# B&R Automation Studio project ZariadenieNaPreklapanieRotorov
Automation Studio 4.7.6.114 SP; Default project

## Configuration Config1

CPU 4PPC30.043F-21B, AutomationRuntime D4.73, Build 6.3.0, Vc V4.72.5

### Task classes (Cpu.sw)
```
Cyclic#3 (cycle 50000 us, tolerance 50000 us):
  Blikanie10 <- Blikace.Blikanie100ms.prg
Cyclic#4 (cycle 100000 us, tolerance 100000 us):
  Blikanie20 <- Blikace.Blikanie200ms.prg
  DatumCasPL <- DatumCasPLC.DatumCasPLC.prg
  Main <- Program.Main.prg
  Preklapac <- Program.Preklapac.prg
  Alarmy <- Program.Alarmy.prg
  OvladanieV <- HMI.OvladanieVizu.prg
Cyclic#5 (cycle 250000 us, tolerance 250000 us):
  Blikanie50 <- Blikace.Blikanie500ms.prg
Cyclic#7 (cycle 1000000 us, tolerance 1000000 us):
  Blikanie1s <- Blikace.Blikanie1s.prg
VcDataObjects: Visu <- HMI.Visu.dob
Binaries: vcctext, arialbd, vccshape, vcchspot, vcnet, vcdsloc, vcbclass, vcfntttf, vccovl, vctcal, Visu03, vcshared, vcpd335x, vcpkat, vcpk, vccbmp, TCData, vcfile, vccbtn, vcmgr, vccdt, vcptelo, vcalarm, Visu01, vccnum, vcpdsw, FWRules, vcrt, arial, udbdef, vcpfppct, vcgclass, vcpdvnc, vccalarm, vccstr, vcdsint, vccbar, Visu02, Role, arconfig, User, asfw, ashwd, ashwac, sysconf, iomap
Libraries: IecCheck, SC, sys_lib, AsBrStr, Runtime, asieccon, fileio, dataobj, astime, standard, vcresman
```

### Hardware
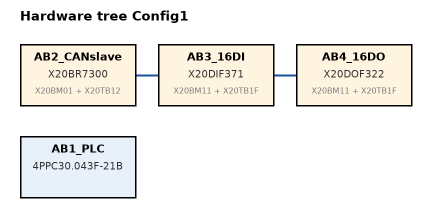
```
AB1_PLC : 4PPC30.043F-21B v1.1.3.0
  Connector IF3:
    ActivateDevice = 1
    Mode = Manual
    InternetAddress = 192.168.1.2
    SubnetMask = 255.255.255.0
    InaNodeNumber = 0
    Vnc1
    VncVcObjectName1 = Visu
    VncKeyMappingFile1 = VC\PS2-Keyboard.dis
    VncMaxConnections1 = 2
    VncRefreshRate1 = 100
  ConfigurationID = ZariadenieNaPreklapanieRotorov_Config1
  PermanentPvSize = 500
  TimerDeviceType = SWIOTIMER
  Cyclic1Duration = 1000
  Cyclic1Tolerance = 0
  Cyclic2Duration = 20000
  Cyclic2Tolerance = 20000
  Cyclic3Duration = 50000
  Cyclic3Tolerance = 50000
  Cyclic4Duration = 100000
  Cyclic4Tolerance = 100000
  Cyclic5Duration = 250000
  Cyclic5Tolerance = 250000
  Cyclic6Duration = 500000
  Cyclic6Tolerance = 500000
  Cyclic7Duration = 1000000
  Cyclic7Tolerance = 1000000
  Cyclic8Duration = 10000
  Cyclic8Tolerance = 30000000
  TimeZone = 145
  VcObjectName = Visu
  RotationAngle = 180
  KeyMappingFile = VC\4PPC30_043F_21B.dis
AB2_CANslave : X20BR7300 v1.4.0.0  [CAN1 -> AB1_PLC.IF4; SL -> X20BM01.SL1; SS1 -> X20TB12.SS]
  Supervision = off
AB3_16DI : X20DIF371 v1.1.0.0  [SS1 -> X20TB1F.SS; SL -> X20BM11.SL1]
  FunctionModel = CANIOBusController
  Supervision = off
AB4_16DO : X20DOF322 v1.4.0.0  [SS1 -> X20TB1F1.SS; SL -> X20BM11a.SL1]
  FunctionModel = CANIOBusController
  Supervision = off
X20BM01 : X20BM01 v2.1.0.0
X20BM11 : X20BM11 v1.0.0.1  [X2X1 -> X20BM01.IF1]
X20BM11a : X20BM11 v1.0.0.1  [X2X1 -> X20BM11.X2X2]
X20TB12 : X20TB12 v1.0.0.0
X20TB1F : X20TB1F v1.0.0.0
X20TB1F1 : X20TB1F v1.0.0.0
```

### IoMap.iom - AB1_PLC/IoMap.iom
```iecst
VAR_CONFIG
	Hardware.KartaAB2_CANSlave_OK AT %IX."AB2_CANslave".IF1.ST1.ModuleOk;
	Hardware.KartaAB3_16DI_OK AT %IX."AB3_16DI".ModuleOk;
	Hardware.KartaAB4_16DO_OK AT %IX."AB4_16DO".ModuleOk;
	Cyclic#1.Zariadenie.IN.TlakVzduchu_OK_S1 AT %IX."AB3_16DI".DigitalInput01;
	Cyclic#1.Preklapac.IN.VstupnyDotlacac_VYSUNUTY_MS1 AT %IX."AB3_16DI".DigitalInput02;
	Cyclic#1.Preklapac.IN.VstupnyDotlacac_ZASUNUTY_MS2 AT %IX."AB3_16DI".DigitalInput03;
	Cyclic#1.Preklapac.IN.VystupnyDotlacac_VYSUNUTY_MS3 AT %IX."AB3_16DI".DigitalInput04;
	Cyclic#1.Preklapac.IN.VystupnyDotlacac_ZASUNUTY_MS4 AT %IX."AB3_16DI".DigitalInput05;
	Cyclic#1.Preklapac.IN.Vytah_HornaPoloha_MS5 AT %IX."AB3_16DI".DigitalInput06;
	Cyclic#1.Preklapac.IN.Vytah_SpodnaPoloha_MS6 AT %IX."AB3_16DI".DigitalInput07;
	Cyclic#1.Preklapac.IN.VstupnyDotlacac_PritomRotora_IS1 AT %IX."AB3_16DI".DigitalInput08;
	Cyclic#1.Zariadenie.IN.Safety_SpatnaVazba_KF1 AT %IX."AB3_16DI".DigitalInput09;
	Cyclic#1.Preklapac.IN.Vytah_Pozicia1_PritomRotora_OS1 AT %IX."AB3_16DI".DigitalInput11;
	Cyclic#1.Preklapac.IN.Vytah_Pozicia2_PritomRotora_OS2 AT %IX."AB3_16DI".DigitalInput12;
	Cyclic#1.Preklapac.IN.VystupnyDopravnik_PLNY_OS3 AT %IX."AB3_16DI".DigitalInput13;
	Cyclic#1.Zariadenie.OUT.Majak_ZeleneSvetlo AT %QX."AB4_16DO".DigitalOutput01;
	Cyclic#1.Zariadenie.OUT.Majak_ZlteSvetlo AT %QX."AB4_16DO".DigitalOutput02;
	Cyclic#1.Zariadenie.OUT.Majak_CerveneSvetlo AT %QX."AB4_16DO".DigitalOutput03;
	Cyclic#1.Zariadenie.OUT.Majak_Hukacka AT %QX."AB4_16DO".DigitalOutput04;
	Cyclic#1.Zariadenie.OUT.Safety_RESET AT %QX."AB4_16DO".DigitalOutput05;
	Cyclic#1.Preklapac.OUT.VstupnyDotlacac_VYSUN_YV1 AT %QX."AB4_16DO".DigitalOutput06;
	Cyclic#1.Preklapac.OUT.VstupnyDotlacac_ZASUN_YV2 AT %QX."AB4_16DO".DigitalOutput07;
	Cyclic#1.Preklapac.OUT.VystupnyDotlacac_VYSUN_YV3 AT %QX."AB4_16DO".DigitalOutput08;
	Cyclic#1.Preklapac.OUT.Vytah_ZDVIH_YV5 AT %QX."AB4_16DO".DigitalOutput10;
	Cyclic#1.Preklapac.OUT.Vytah_ZOSTUP_YV6 AT %QX."AB4_16DO".DigitalOutput11;
	Cyclic#1.Zariadenie.IN.Safety_SpatnaVazba_Ventil_YVS1 AT %IX."AB3_16DI".DigitalInput14;
	Cyclic#1.Zariadenie.IN.Safety_SpatnaVazba_Ventil_YVS2 AT %IX."AB3_16DI".DigitalInput15;
	Cyclic#1.Zariadenie.IN.Safety_Aktivne AT %IX."AB3_16DI".DigitalInput16;
	Cyclic#1.Preklapac.IN.VystupnyDopravnik_StavOK AT %IX."AB3_16DI".DigitalInput10;
END_VAR
```

- Physical/Config1/AB1_PLC/PvMap.vvm: same as Physical/Config1/AB1_PLC/Cpu.per
## Logical view

Binary libraries used (declarations not repeated): RUNTIME, OPERATOR, AsIecCon, astime, standard, AsBrStr, FileIO, sys_lib

### Global.typ - Global data types
```iecst
(********************************************************************
 * COPYRIGHT -- Microsoft
 ********************************************************************
 * File: Global.typ
 * Author: Martin
 * Created: February 11, 2016
 ********************************************************************
 * Global data types of project Zamazat_1
 ********************************************************************)
(**************Stav hardware*****************************)

TYPE
	HardwareSTAV_typ : 	STRUCT
		KartaAB2_CANSlave_OK : BOOL;
		KartaAB3_16DI_OK : BOOL;
		KartaAB4_16DO_OK : BOOL;
	END_STRUCT;
END_TYPE

(**************************Vizualizacia**********************************************)

TYPE
	Vizu_typ : 	STRUCT
		CisloAktualnejObrazovky : USINT;
		CisloZadanejObrazovky : USINT;
		TL_RezimAutomat : BOOL;
		StavZariadenia_Farba : USINT;
		StavZariadenia_Index : USINT;
		TL_RezimManual_DISABLE : BOOL; (*0 - odomknuté, 1 - zamknuté*)
		TL_StartAutomat_DISABLE : BOOL;
		TL_UkoncenieCyklu_DISABLE : BOOL;
		TL_Reset_DISABLE : BOOL;
		TL_RR_PreklapacDotlacace_DISABLE : BOOL;
		TL_RR_PreklapacZdvih_DISABLE : BOOL;
		Slider : USINT;
		FarbaTlacitkaAlarm_Index : BOOL;
		ZobrazSymbolAlarmu : BOOL;
		TP_PopUp_ResetZariadenia : USINT;
		TP_PopUp_VystupDopRozpojeny : USINT;
		PodsvietenieTlacitka_ResetCS : USINT;
	END_STRUCT;
END_TYPE

(**************************Pracovisko************************************************)

TYPE
	Zariadenie_typ : 	STRUCT
		IN : ZariadenieIN_typ;
		OUT : ZariadenieOUT_typ;
		PAR : ZariadeniePAR_typ;
		STAV : ZariadenieSTAV_typ;
		Automat : BOOL;
		Manual : BOOL;
		Reset : BOOL;
		KoniecCyklu : BOOL;
		Majak_HukackaON : BOOL;
	END_STRUCT;
	ZariadenieIN_typ : 	STRUCT
		TlakVzduchu_OK_S1 : BOOL;
		Safety_SpatnaVazba_KF1 : BOOL;
		Safety_ReleCakaNaReset_KF1 : BOOL;
		Safety_SpatnaVazba_Ventil_YVS1 : BOOL;
		Safety_SpatnaVazba_Ventil_YVS2 : BOOL;
		Safety_Aktivne : BOOL;
	END_STRUCT;
	ZariadenieOUT_typ : 	STRUCT
		Majak_ZeleneSvetlo : BOOL;
		Majak_ZlteSvetlo : BOOL;
		Majak_CerveneSvetlo : BOOL;
		Majak_Hukacka : BOOL;
		Safety_RESET : BOOL;
	END_STRUCT;
	ZariadeniePAR_typ : 	STRUCT
		PAR_0 : USINT;
	END_STRUCT;
	ZariadenieSTAV_typ : 	STRUCT
		Automat : BOOL;
		Manual : BOOL;
		PoINIT : BOOL;
		READY_TO_START : BOOL;
		UkoncenieCyklu_BUSY : BOOL;
		Hardware_OK : BOOL;
	END_STRUCT;
END_TYPE

(***************Preklapač*************************************)

TYPE
	Preklapac_typ : 	STRUCT
		IN : PreklapacIN_typ;
		OUT : PreklapacOUT_typ;
		PAR : PreklapacPAR_typ;
		STAV : PreklapacSTAV_typ;
		Automat : BOOL;
		Manual : BOOL;
		Reset : BOOL;
		KoniecCyklu : BOOL;
	END_STRUCT;
	PreklapacIN_typ : 	STRUCT
		VstupnyDotlacac_VYSUNUTY_MS1 : BOOL;
		VstupnyDotlacac_ZASUNUTY_MS2 : BOOL;
		VstupnyDotlacac_PritomRotora_IS1 : BOOL;
		VystupnyDotlacac_VYSUNUTY_MS3 : BOOL;
		VystupnyDotlacac_ZASUNUTY_MS4 : BOOL;
		Vytah_HornaPoloha_MS5 : BOOL;
		Vytah_SpodnaPoloha_MS6 : BOOL;
		Vytah_Pozicia1_PritomRotora_OS1 : BOOL;
		Vytah_Pozicia2_PritomRotora_OS2 : BOOL;
		VystupnyDopravnik_PLNY_OS3 : BOOL;
		VystupnyDopravnik_StavOK : BOOL;
	END_STRUCT;
	PreklapacOUT_typ : 	STRUCT
		VstupnyDotlacac_VYSUN_YV1 : BOOL;
		VstupnyDotlacac_ZASUN_YV2 : BOOL;
		VystupnyDotlacac_VYSUN_YV3 : BOOL;
		Vytah_ZDVIH_YV5 : BOOL;
		Vytah_ZOSTUP_YV6 : BOOL;
	END_STRUCT;
	PreklapacPAR_typ : 	STRUCT
		PAR_0 : USINT;
	END_STRUCT;
	PreklapacSTAV_typ : 	STRUCT
		PoINIT : BOOL;
	END_STRUCT;
END_TYPE
```

### Global.var - Global variables
```iecst
(********************************************************************
 * COPYRIGHT -- Microsoft
 ********************************************************************
 * File: Global.var
 * Author: Martin
 * Created: February 11, 2016
 ********************************************************************
 * Global variables of project Zamazat_1
 ********************************************************************)
(******************Blikače*****************************)
VAR
	Blikac100ms : BOOL;
	Blikac200ms : BOOL;
	Blikac500ms : BOOL;
	Blikac1s : BOOL;
END_VAR
(**********Nastavenie času**************)
VAR
	DTSetTime_0 : DTSetTime := (0);
	DTGetTime_0 : DTGetTime := (0);
END_VAR
(*****************Alarmy*****************************)
VAR
	Alarmy : ARRAY[0..100] OF BOOL;
	NastalaPorucha : BOOL;
	PotvrdenieAlarmov : BOOL;
END_VAR
(*************Všeobecné premenné*************)
VAR
	Hardware : HardwareSTAV_typ := (0);
	Zariadenie : Zariadenie_typ := (0);
	Vizu : Vizu_typ := (0);
	Preklapac : Preklapac_typ := (0);
	SC_Preklapac : SequenceControlTyp := (0);
END_VAR
```

### Package Logical/Libraries - Global libraries

### Library Logical/Libraries/SC (IEC)

#### Types.typ - Exported data types
```iecst
TYPE
	SequenceControlTyp : 	STRUCT
		StepName : STRING[200];
		Step : UINT;
		Switch1 : BOOL;
		Switch2 : BOOL;
		Switch3 : BOOL;
		ResetStep : BOOL;
		LastStep : BOOL;
		IdleTime : TON;
		AlarmTime : TON;
	END_STRUCT;
END_TYPE
```

#### SC.fun - Exported functions and function blocks
```iecst
FUNCTION SequenceControl : BOOL
	VAR_IN_OUT
		SC : SequenceControlTyp;
	END_VAR
END_FUNCTION
```

#### SequenceControl.st
```iecst
(* TODO: Add your comment here *)
FUNCTION SequenceControl

	IF SC.ResetStep THEN
		brsmemset(ADR(SC.StepName),0,SIZEOF(SC.StepName));
		SC.Switch1:= FALSE;
		SC.Switch2:= FALSE;
		SC.Switch3:= FALSE;
		SC.IdleTime.IN:= FALSE;
		SC.AlarmTime.IN:= FALSE;
		SC.ResetStep:= FALSE;
	END_IF

	IF SC.LastStep THEN
		brsmemset(ADR(SC.StepName),0,SIZEOF(SC.StepName));
		SC.Switch1:= FALSE;
		SC.Switch2:= FALSE;
		SC.Switch3:= FALSE;
		SC.IdleTime.IN:= FALSE;
		SC.AlarmTime.IN:= FALSE;
		SC.Step:= 0;
		SC.LastStep:= FALSE;
	END_IF

	//Volanie časovačov//
	SC.AlarmTime();
	SC.IdleTime();

END_FUNCTION
```

### Library Logical/Libraries/IecCheck (IEC)
Depends on: sys_lib, AsBrStr

#### IecCheck.fun - Exported functions and function blocks
```iecst
FUNCTION CheckDivSint : SINT (* Check divisor for SINT division *)
	VAR_INPUT
		divisor : SINT;
	END_VAR
END_FUNCTION

FUNCTION CheckDivUsint : USINT (* Check divisor for USINT division *)
	VAR_INPUT
		divisor : USINT;
	END_VAR
END_FUNCTION

FUNCTION CheckDivInt : INT (* Check divisor for INT division *)
	VAR_INPUT
		divisor : INT;
	END_VAR
END_FUNCTION

FUNCTION CheckDivUint : UINT (* Check divisor for UINT division *)
	VAR_INPUT
		divisor : UINT;
	END_VAR
END_FUNCTION

FUNCTION CheckDivDint : DINT (* Check divisor for DINT division *)
	VAR_INPUT
		divisor : DINT;
	END_VAR
END_FUNCTION

FUNCTION CheckDivUdint : UDINT (* Check divisor for UDINT division *)
	VAR_INPUT
		divisor : UDINT;
	END_VAR
END_FUNCTION

FUNCTION CheckDivReal : REAL (* Check divisor for REAL division *)
	VAR_INPUT
		divisor : REAL;
	END_VAR
END_FUNCTION

FUNCTION CheckDivLReal : LREAL (* Check divisor for LREAL division, not available for SG3 and SGC *)
	VAR_INPUT
		divisor : LREAL;
	END_VAR
END_FUNCTION

FUNCTION CheckBounds : DINT (* Check range for array access *)
	VAR_INPUT
		index : DINT;
		lower : DINT;
		upper : DINT;
	END_VAR
END_FUNCTION

FUNCTION CheckRange : DINT (* Check range for enumeration *)
	VAR_INPUT
		value : DINT;
		lower : DINT;
		upper : DINT;
	END_VAR
END_FUNCTION

FUNCTION CheckSignedSubrange : DINT (* Check range for subrange of signed data types *)
	VAR_INPUT
		value : DINT;
		lower : DINT;
		upper : DINT;
	END_VAR
END_FUNCTION

FUNCTION CheckUnsignedSubrange : UDINT (* Check range for subrange of unsigned data types *)
	VAR_INPUT
		value : UDINT;
		lower : UDINT;
		upper : UDINT;
	END_VAR
END_FUNCTION

FUNCTION CheckReadAccess : UDINT (* Check address when reading dynamic variables *)
	VAR_INPUT
		address : UDINT;
	END_VAR
END_FUNCTION

FUNCTION CheckWriteAccess : UDINT (* Check address when writing dynamic variables *)
	VAR_INPUT
		address : UDINT;
	END_VAR
END_FUNCTION

FUNCTION MakeEntry : UDINT (* Makes an entry (log book entry) in the error log book *)
	VAR
		taskname : STRING[30];
		group : USINT;
		status_name : UINT;
		out_text : STRING[80];
	END_VAR
	VAR_INPUT
		number : UINT;
		index : DINT;
		text : STRING[50];
	END_VAR
END_FUNCTION
```

#### IecCheck.st - Implementation file
```iecst
(* Check divisor for SINT division *)
FUNCTION CheckDivSint
	IF divisor=0 THEN
		CheckDivSint:=1;
		MakeEntry(55555,divisor,'CheckDivSint');
	ELSE
		CheckDivSint:=divisor;
	END_IF
END_FUNCTION

(* Check divisor for USINT division *)
FUNCTION CheckDivUsint
	IF divisor=0 THEN
		CheckDivUsint:=1;
		MakeEntry(55555,divisor,'CheckDivUsint');
	ELSE
		CheckDivUsint:=divisor;
	END_IF
END_FUNCTION

(* Check divisor for INT division *)
FUNCTION CheckDivInt
	IF divisor=0 THEN
		CheckDivInt:=1;
		MakeEntry(55555,divisor,'CheckDivInt');
	ELSE
		CheckDivInt:=divisor;
	END_IF
END_FUNCTION

(* Check divisor for UINT division *)
FUNCTION CheckDivUint
	IF divisor=0 THEN
		CheckDivUint:=1;
		MakeEntry(55555,divisor,'CheckDivUint');
	ELSE
		CheckDivUint:=divisor;
	END_IF
END_FUNCTION

(* Check divisor for DINT division *)
FUNCTION CheckDivDint
	IF divisor=0 THEN
		CheckDivDint:=1;
		MakeEntry(55555,divisor,'CheckDivDint');
	ELSE
		CheckDivDint:=divisor;
	END_IF
END_FUNCTION

(* Check divisor for UDINT division *)
FUNCTION CheckDivUdint
	IF divisor=0 THEN
		CheckDivUdint:=1;
		MakeEntry(55555,divisor,'CheckDivUdint');
	ELSE
		CheckDivUdint:=divisor;
	END_IF
END_FUNCTION

(* Check divisor for REAL division *)
FUNCTION CheckDivReal
	IF divisor=0 THEN
		CheckDivReal:=1;
		MakeEntry(55555,0,'CheckDivReal');
	ELSE
		CheckDivReal:=divisor;
	END_IF
END_FUNCTION

(* Check divisor for LREAL division *)
FUNCTION CheckDivLReal
	IF divisor=0 THEN
		CheckDivLReal:=1;
		MakeEntry(55555,0,'CheckDivLReal');
	ELSE
		CheckDivLReal:=divisor;
	END_IF
END_FUNCTION

(* Check range for array access *)
FUNCTION CheckBounds
	IF index < lower THEN
		CheckBounds := lower;
		MakeEntry(55555,index,'CheckBounds');
	ELSIF index > upper THEN
		CheckBounds := upper;
		MakeEntry(55555,index,'CheckBounds');
	ELSE
		CheckBounds := index;
	END_IF
END_FUNCTION

(* Check range for enumeration *)
FUNCTION CheckRange
	IF value < lower THEN
		CheckRange := lower;
		MakeEntry(55555,value,'CheckRange');
	ELSIF value > upper THEN
		CheckRange := upper;
		MakeEntry(55555,value,'CheckRange');
	ELSE
		CheckRange := value;
	END_IF
END_FUNCTION

(* Check range for subrange of signed data types *)
FUNCTION CheckSignedSubrange
	IF value < lower THEN
		CheckSignedSubrange := lower;
		MakeEntry(55555,value,'CheckSignedSubrange');
	ELSIF value > upper THEN
		CheckSignedSubrange := upper;
		MakeEntry(55555,value,'CheckSignedSubrange');
	ELSE
		CheckSignedSubrange := value;
	END_IF
END_FUNCTION

(* Check range for subrange of unsigned data types *)
FUNCTION CheckUnsignedSubrange
	IF value < lower THEN
		CheckUnsignedSubrange := lower;
		MakeEntry(55555,value,'CheckUnsignedSubrange');
	ELSIF value > upper THEN
		CheckUnsignedSubrange := upper;
		MakeEntry(55555,value,'CheckUnsignedSubrange');
	ELSE
		CheckUnsignedSubrange := value;
	END_IF
END_FUNCTION

(* Check address when reading dynamic variables *)
FUNCTION CheckReadAccess
	IF address=0 THEN
		(* TODO: Insert an appropriate code, see AutomationStudio help for further information *)
		MakeEntry(55555,address,'Read from NULL');
	END_IF

	CheckReadAccess:=0;
END_FUNCTION

(* Check address when writing dynamic variables *)
FUNCTION CheckWriteAccess
	IF address=0 THEN
		(* TODO: Insert an appropriate code, see AutomationStudio help for further information *)
		MakeEntry(55555,address,'Write to NULL');
	END_IF

	CheckWriteAccess:=0;
END_FUNCTION

(* Makes an entry (log book entry) in the error log book *)
FUNCTION MakeEntry
		status_name := ST_name(0,ADR(taskname),ADR(group));

		brsstrcpy(ADR(out_text),ADR(text));
		brsstrcat(ADR(out_text),ADR(' > in task > '));
  		brsstrcat(ADR(out_text),ADR(taskname));
		MakeEntry := ADR(out_text);
		ERRxfatal(number,index,ADR(out_text));
END_FUNCTION
```

### Package Logical/Program - Riadiace programy

### Program Logical/Program/Main (IEC)

#### Main.st - Init, cyclic, exit code
```iecst
PROGRAM _INIT

END_PROGRAM

PROGRAM _CYCLIC

    //****************************************Príznak hardware pracoviska OK***********************************//

    IF Hardware.KartaAB2_CANSlave_OK
        AND Hardware.KartaAB3_16DI_OK
        AND Hardware.KartaAB4_16DO_OK THEN
        Zariadenie.STAV.Hardware_OK:= TRUE;
    ELSE
        Zariadenie.STAV.Hardware_OK:= FALSE;
    END_IF

    //***************************************Ovládanie majáka**************************************************//
    //Zelene svetlo//
    IF Zariadenie.STAV.Automat THEN
        Zariadenie.OUT.Majak_ZeleneSvetlo:= TRUE;
    ELSIF Zariadenie.STAV.Manual THEN
        Zariadenie.OUT.Majak_ZeleneSvetlo:= Blikac500ms;
    ELSE
        Zariadenie.OUT.Majak_ZeleneSvetlo:= FALSE;
    END_IF

    //Žlté svetlo//
    IF Zariadenie.STAV.Automat AND NOT Zariadenie.STAV.PoINIT THEN
        Zariadenie.OUT.Majak_ZlteSvetlo:= Blikac500ms;
    ELSE
        Zariadenie.OUT.Majak_ZlteSvetlo:= FALSE;
    END_IF

    //Červené svetlo//
    IF NastalaPorucha THEN
        Zariadenie.OUT.Majak_CerveneSvetlo:= TRUE;
    ELSIF NOT Zariadenie.IN.Safety_Aktivne THEN
        Zariadenie.OUT.Majak_CerveneSvetlo:= TRUE;
    ELSE
        Zariadenie.OUT.Majak_CerveneSvetlo:= FALSE;
    END_IF

    //Húkačka//
    IF EDGEPOS(NastalaPorucha) THEN
        Zariadenie.Majak_HukackaON:= TRUE;
    END_IF

    IF Zariadenie.Majak_HukackaON THEN
        Zariadenie.OUT.Majak_Hukacka:= Blikac500ms;
    ELSE
        Zariadenie.OUT.Majak_Hukacka:= FALSE;
    END_IF

    //**************************************Ukončenie pracovného cyklu na pracovisku**********************************************//
    IF Zariadenie.KoniecCyklu THEN
        Zariadenie.STAV.UkoncenieCyklu_BUSY:= TRUE;
        IF Preklapac.Automat THEN
            Preklapac.KoniecCyklu:= TRUE;
        END_IF
        Zariadenie.KoniecCyklu:= FALSE;
    END_IF

    IF NOT Zariadenie.STAV.Automat THEN
        Zariadenie.STAV.UkoncenieCyklu_BUSY:= FALSE;
    END_IF

    //****************************************Resetovanie pracoviska****************************************************************//
    //Normálne//
    IF Zariadenie.Reset THEN
        Preklapac.Reset:= TRUE;
        Zariadenie.Reset:= FALSE;
    END_IF

    //Pri stlačení tlačítka Automat//
    IF Vizu.TL_RezimAutomat THEN
        IF Zariadenie.STAV.Manual THEN
            Zariadenie.Reset:= TRUE;
        END_IF
        Vizu.TL_RezimAutomat:= FALSE;
    END_IF

    //**************************************Manuálny režim pracoviska*************************************************************//
    IF Zariadenie.Manual THEN
        Preklapac.Manual:= TRUE;
        Zariadenie.Manual:= FALSE;
    END_IF

    //Príznak je zvolený režim Manuál//
    IF Preklapac.Manual THEN
        Zariadenie.STAV.Manual:= TRUE;
    ELSE
        Zariadenie.STAV.Manual:= FALSE;
    END_IF

    //***************************************Automatický režim pracoviska**********************************************************//
    IF Zariadenie.Automat THEN
        IF Zariadenie.STAV.Hardware_OK THEN
            Preklapac.Automat:= TRUE;
        END_IF
        Zariadenie.Automat:= FALSE;
    END_IF

    //Príznak je zvolený režim Automat//
    IF Preklapac.Automat THEN
        Zariadenie.STAV.Automat:= TRUE;
    ELSE
        Zariadenie.STAV.Automat:= FALSE;
    END_IF

    //Príznak Zariadenie je po inicializácii//
    IF Preklapac.STAV.PoINIT THEN
        Zariadenie.STAV.PoINIT:= TRUE;
    ELSE
        Zariadenie.STAV.PoINIT:= FALSE;
    END_IF

    //****************************************Príznak Zariadenie pripravené na spustenie********************************************//
    IF SC_Preklapac.Step = 1 THEN
        Zariadenie.STAV.READY_TO_START:= TRUE;
    ELSE
        Zariadenie.STAV.READY_TO_START:= FALSE;
    END_IF

END_PROGRAM

PROGRAM _EXIT
	(* Insert code here *)

END_PROGRAM
```

### Program Logical/Program/Preklapac (IEC)

#### Main.st - Init, cyclic, exit code
```iecst
PROGRAM _INIT
	(* Insert code here *)

END_PROGRAM

PROGRAM _CYCLIC

    //Volanie funkcie SequenceControl//
    SequenceControl(SC:= SC_Preklapac);

    //Volanie podprogramov//
    VstupnyDotlacac;
    Zdvih;
    VystupnyDotlacac;

    //Reset sekcie //
    IF NOT Zariadenie.IN.Safety_Aktivne THEN
		SC_Preklapac.Step:= 0;
	ELSIF NastalaPorucha THEN
        SC_Preklapac.Step:= 0;
    ELSIF Preklapac.Reset THEN
        SC_Preklapac.Step:= 0;
    END_IF

    CASE SC_Preklapac.Step OF

        0:
            SC_Preklapac.StepName:='0 - Nulovanie';
            Preklapac.Automat:= FALSE;
            Preklapac.KoniecCyklu:= FALSE;
            Preklapac.Manual:= FALSE;
            Preklapac.Reset:= FALSE;
            Preklapac.STAV.PoINIT:= FALSE;
            SC_VstupnyDotlacac.Step:= 0;
            SC_Zdvih.Step:= 0;
            SC_VystupnyDotlacac.Step:= 0;

            IF Zariadenie.IN.Safety_Aktivne AND NOT NastalaPorucha THEN
                SC_Preklapac.ResetStep:= TRUE;
                SC_Preklapac.Step:= 1;
            END_IF

        1:
            SC_Preklapac.StepName:='1 - Cakam na spustenie vyroby';
            IF Preklapac.Automat THEN
                SC_Preklapac.Step:= 2;
            ELSIF Preklapac.Manual THEN
                SC_Preklapac.Step:= 700;
            END_IF

        //********************************************************Inicializácia****************************************************************************//

        2:
            SC_Preklapac.StepName:='2 - Inicializacia - cakam na spustenie inicializacie';
            SC_Preklapac.IdleTime.PT:= T#500ms;
            SC_Preklapac.AlarmTime.PT:= T#5s;

            SC_Preklapac.IdleTime.IN:= TRUE;

            IF SC_Preklapac.IdleTime.Q THEN
                SC_Preklapac.ResetStep:= TRUE;
                SC_Preklapac.Step:= 3;
            END_IF

        3:
            SC_Preklapac.StepName:='3 - Inicializacia - cakam na zasunutie vstupneho a vystupneho dotlacaca';
            SC_Preklapac.IdleTime.PT:= T#500ms;
            SC_Preklapac.AlarmTime.PT:= T#5s;

            IF NOT SC_Preklapac.Switch1 THEN
                VstupnyDotlacac_ZASUN:= TRUE;
                VystupnyDotlacac_ZASUN:= TRUE;
                SC_Preklapac.Switch1:= TRUE;
            END_IF

            IF Preklapac.IN.VstupnyDotlacac_ZASUNUTY_MS2 AND Preklapac.IN.VystupnyDotlacac_ZASUNUTY_MS4 THEN
                SC_Preklapac.ResetStep:= TRUE;
                SC_Preklapac.Step:= 5;
            END_IF

        5:
            SC_Preklapac.StepName:='5 - Inicializacia - cakam na presun zdvihu do spodnej polohy';
            SC_Preklapac.IdleTime.PT:= T#500ms;
            SC_Preklapac.AlarmTime.PT:= T#5s;

            IF NOT SC_Preklapac.Switch1 THEN
                Zdvih_ZASUN:= TRUE;
                SC_Preklapac.Switch1:= TRUE;
            END_IF

            IF Preklapac.IN.Vytah_SpodnaPoloha_MS6 THEN
                SC_Preklapac.ResetStep:= TRUE;
                SC_Preklapac.Step:= 10;
            END_IF

        10:
            SC_Preklapac.StepName:='10 - Inicializacia - kontrolujem pritomnost rotorov na zdvihu';
            SC_Preklapac.IdleTime.PT:= T#500ms;
            SC_Preklapac.AlarmTime.PT:= T#5s;

            IF Preklapac.IN.Vytah_Pozicia1_PritomRotora_OS1 OR Preklapac.IN.Vytah_Pozicia2_PritomRotora_OS2 THEN
                Preklapac.STAV.PoINIT:= TRUE;
                SC_Preklapac.ResetStep:= TRUE;
                SC_Preklapac.Step:= 115;
            ELSE
                Preklapac.STAV.PoINIT:= TRUE;
                SC_Preklapac.ResetStep:= TRUE;
                SC_Preklapac.Step:= 100;
            END_IF

            //********************************************************Automatický režim****************************************************************************//

        100:
            SC_Preklapac.StepName:='100 - Automaticky Rezim - cakam na prichod rotora';
            SC_Preklapac.IdleTime.PT:= T#300ms;
            SC_Preklapac.AlarmTime.PT:= T#5s;

            SC_Preklapac.IdleTime.IN:= Preklapac.IN.VstupnyDotlacac_PritomRotora_IS1;

            IF Preklapac.KoniecCyklu THEN
                SC_Preklapac.ResetStep:= TRUE;
				SC_Preklapac.Step:= 0;
			ELSIF NOT Preklapac.IN.VystupnyDopravnik_StavOK THEN
				SC_Preklapac.Step:= 0;
            ELSIF SC_Preklapac.IdleTime.Q THEN
                SC_Preklapac.ResetStep:= TRUE;
                SC_Preklapac.Step:= 108;
            END_IF

        108:
            SC_Preklapac.StepName:='108 - Automaticky Rezim - cakam na vysunutie vstupneho dotlacaca';
            SC_Preklapac.IdleTime.PT:= T#100ms;
            SC_Preklapac.AlarmTime.PT:= T#5s;

            SC_Preklapac.IdleTime.IN:= Preklapac.IN.VstupnyDotlacac_VYSUNUTY_MS1;

            IF NOT SC_Preklapac.Switch1 AND Preklapac.IN.Vytah_SpodnaPoloha_MS6 THEN
                VstupnyDotlacac_VYSUN:= TRUE;
                SC_Preklapac.Switch1:= TRUE;
            END_IF

            IF Preklapac.IN.VstupnyDotlacac_VYSUNUTY_MS1 AND SC_Preklapac.IdleTime.Q THEN
                SC_Preklapac.ResetStep:= TRUE;
                SC_Preklapac.Step:= 115;
            END_IF

		115:
			SC_Preklapac.StepName:='115 - Automaticky Rezim - kontrolujem pocet kusov na zdvihu';
			SC_Preklapac.IdleTime.PT:= T#500ms;
			SC_Preklapac.AlarmTime.PT:= T#5s;

			IF Preklapac.IN.Vytah_Pozicia1_PritomRotora_OS1 AND Preklapac.IN.Vytah_Pozicia2_PritomRotora_OS2 THEN
				SC_Preklapac.ResetStep:= TRUE;
				SC_Preklapac.Step:= 120;
			ELSE
				SC_Preklapac.ResetStep:= TRUE;
				SC_Preklapac.Step:= 118;
			END_IF

		118:
			SC_Preklapac.StepName:='118 - Automaticky Rezim - cakam na zasunutie vstupneho dotlacaca';
			SC_Preklapac.IdleTime.PT:= T#500ms;
			SC_Preklapac.AlarmTime.PT:= T#5s;

			IF NOT SC_Preklapac.Switch1 THEN
				VstupnyDotlacac_ZASUN:= TRUE;
				SC_Preklapac.Switch1:= TRUE;
			END_IF

			IF Preklapac.IN.VstupnyDotlacac_ZASUNUTY_MS2 THEN
				SC_Preklapac.ResetStep:= TRUE;
				SC_Preklapac.Step:= 100;
			END_IF

        120:
            SC_Preklapac.StepName:='120 - Automaticky Rezim - cakam na presun zdvihu do hornej polohy';
            SC_Preklapac.IdleTime.PT:= T#100ms;
            SC_Preklapac.AlarmTime.PT:= T#5s;

            SC_Preklapac.IdleTime.IN:= Preklapac.IN.Vytah_HornaPoloha_MS5;

            IF NOT SC_Preklapac.Switch1 AND Preklapac.IN.VystupnyDotlacac_ZASUNUTY_MS4 THEN
                Zdvih_VYSUN:= TRUE;
                SC_Preklapac.Switch1:= TRUE;
            END_IF

            IF Preklapac.IN.Vytah_HornaPoloha_MS5 AND SC_Preklapac.IdleTime.Q THEN
                SC_Preklapac.ResetStep:= TRUE;
                SC_Preklapac.Step:= 125;
            END_IF

        125:
            SC_Preklapac.StepName:='125 - Automaticky Rezim - kontrola zaplnenia vystupneho dopravnika';
            SC_Preklapac.IdleTime.PT:= T#200ms;
            SC_Preklapac.AlarmTime.PT:= T#5s;

            SC_Preklapac.AlarmTime.IN:= Preklapac.KoniecCyklu;

            SC_Preklapac.IdleTime.IN:= NOT Preklapac.IN.VystupnyDopravnik_PLNY_OS3 AND Preklapac.IN.VystupnyDopravnik_StavOK;

			IF NOT Preklapac.IN.VystupnyDopravnik_StavOK THEN
				SC_Preklapac.Step:= 0;
            ELSIF SC_Preklapac.IdleTime.Q THEN
                SC_Preklapac.ResetStep:= TRUE;
                SC_Preklapac.Step:= 128;
            ELSIF SC_Preklapac.AlarmTime.Q THEN
                SC_Preklapac.ResetStep:= TRUE;
                SC_Preklapac.Step:= 0;
            END_IF

        128:
            SC_Preklapac.StepName:='128 - Automaticky Rezim - cakam na vysunutie vystupneho dotlacaca';
            SC_Preklapac.IdleTime.PT:= T#100ms;
            SC_Preklapac.AlarmTime.PT:= T#5s;

            SC_Preklapac.IdleTime.IN:= Preklapac.IN.VystupnyDotlacac_VYSUNUTY_MS3;

            IF NOT SC_Preklapac.Switch1 AND Preklapac.IN.Vytah_HornaPoloha_MS5 THEN
                VystupnyDotlacac_VYSUN:= TRUE;
                SC_Preklapac.Switch1:= TRUE;
            END_IF

            IF Preklapac.IN.VystupnyDotlacac_VYSUNUTY_MS3 AND SC_Preklapac.IdleTime.Q THEN
                SC_Preklapac.ResetStep:= TRUE;
                SC_Preklapac.Step:= 130;
            END_IF

        130:
            SC_Preklapac.StepName:='130 - Automaticky Rezim - cakam na zasunutie vystupneho dotlacaca';
            SC_Preklapac.IdleTime.PT:= T#500ms;
            SC_Preklapac.AlarmTime.PT:= T#5s;

            IF NOT SC_Preklapac.Switch1 THEN
                VystupnyDotlacac_ZASUN:= TRUE;
                SC_Preklapac.Switch1:= TRUE;
            END_IF

            IF Preklapac.IN.VystupnyDotlacac_ZASUNUTY_MS4 THEN
                SC_Preklapac.ResetStep:= TRUE;
                SC_Preklapac.Step:= 135;
            END_IF

        135:
            SC_Preklapac.StepName:='135 - Automaticky Rezim - cakam na presun zdvihu do spodnej polohy';
            SC_Preklapac.IdleTime.PT:= T#100ms;
            SC_Preklapac.AlarmTime.PT:= T#5s;

            SC_Preklapac.IdleTime.IN:= Preklapac.IN.Vytah_SpodnaPoloha_MS6;

            IF NOT SC_Preklapac.Switch1 AND Preklapac.IN.VystupnyDotlacac_ZASUNUTY_MS4 THEN
                Zdvih_ZASUN:= TRUE;
                SC_Preklapac.Switch1:= TRUE;
            END_IF

            IF Preklapac.IN.Vytah_SpodnaPoloha_MS6 THEN
                SC_Preklapac.ResetStep:= TRUE;
                SC_Preklapac.Step:= 138;
            END_IF

		138:
			SC_Preklapac.StepName:='138 - Automaticky Rezim - cakam na zasunutie vstupneho dotlacaca';
			SC_Preklapac.IdleTime.PT:= T#500ms;
			SC_Preklapac.AlarmTime.PT:= T#5s;

			IF NOT SC_Preklapac.Switch1 THEN
				VstupnyDotlacac_ZASUN:= TRUE;
				SC_Preklapac.Switch1:= TRUE;
			END_IF

			IF Preklapac.IN.VstupnyDotlacac_ZASUNUTY_MS2 THEN
				SC_Preklapac.ResetStep:= TRUE;
				SC_Preklapac.Step:= 100;
			END_IF

            //*******************************************Manuálny režim***************************************************************//
        700:
            SC_Preklapac.StepName:='700 - Manualny rezim';
			SC_Preklapac.IdleTime.PT:= T#3s;
			SC_Preklapac.AlarmTime.PT:= T#5s;

    END_CASE

END_PROGRAM

PROGRAM _EXIT
	(* Insert code here *)

END_PROGRAM
```

#### Variables.var - Local variables
```iecst
VAR
	SC_VstupnyDotlacac : SequenceControlTyp := (0);
	VstupnyDotlacac_VYSUN : BOOL := FALSE;
	VstupnyDotlacac_ZASUN : BOOL := FALSE;
	SC_Zdvih : SequenceControlTyp := (0);
	Zdvih_VYSUN : BOOL := FALSE;
	Zdvih_ZASUN : BOOL := FALSE;
	SC_VystupnyDotlacac : SequenceControlTyp := (0);
	VystupnyDotlacac_VYSUN : BOOL := FALSE;
	VystupnyDotlacac_ZASUN : BOOL := FALSE;
END_VAR
```

#### VstupnyDotlacac.st
```iecst
ACTION VstupnyDotlacac:

    //Volanie funkcie SequenceControl//
    SequenceControl(SC:= SC_VstupnyDotlacac);

    CASE SC_VstupnyDotlacac.Step OF

        0:
            SC_VstupnyDotlacac.StepName:= '0 - Nulovanie';
            VstupnyDotlacac_VYSUN:= FALSE;
            VstupnyDotlacac_ZASUN:= FALSE;
            Preklapac.OUT.VstupnyDotlacac_VYSUN_YV1:= FALSE;
            Preklapac.OUT.VstupnyDotlacac_ZASUN_YV2:= FALSE;

            IF SC_Preklapac.Step <> 0 THEN
                SC_VstupnyDotlacac.ResetStep:= TRUE;
                SC_VstupnyDotlacac.Step:= 1;
            END_IF

        1:
            SC_VstupnyDotlacac.StepName:= '1 - Rozhodnutie o cinnosti';
            IF VstupnyDotlacac_VYSUN THEN
                SC_VstupnyDotlacac.Step:= 10;
            ELSIF VstupnyDotlacac_ZASUN THEN
                SC_VstupnyDotlacac.Step:= 20;
            END_IF

        10:
            SC_VstupnyDotlacac.StepName:= '10 - Vysunutie dotlacaca';
            SC_VstupnyDotlacac.IdleTime.PT:= T#3s;
            SC_VstupnyDotlacac.AlarmTime.PT:= T#3s;

            IF Preklapac.Automat THEN
                SC_VstupnyDotlacac.AlarmTime.IN:= TRUE;
            ELSE
                SC_VstupnyDotlacac.IdleTime.IN:= TRUE;
            END_IF

            IF NOT SC_VstupnyDotlacac.Switch1 THEN
                Preklapac.OUT.VstupnyDotlacac_ZASUN_YV2:= FALSE;
                Preklapac.OUT.VstupnyDotlacac_VYSUN_YV1:= TRUE;
                SC_VstupnyDotlacac.IdleTime.IN:= TRUE;
                SC_VstupnyDotlacac.Switch1:= TRUE;
            END_IF

            IF Preklapac.IN.VstupnyDotlacac_VYSUNUTY_MS1 OR SC_VstupnyDotlacac.IdleTime.Q THEN
                SC_VstupnyDotlacac.ResetStep:= TRUE;
                SC_VstupnyDotlacac.Step:= 0;
            ELSIF SC_VstupnyDotlacac.AlarmTime.Q THEN
                SC_VstupnyDotlacac.ResetStep:= TRUE;
                SC_VstupnyDotlacac.Step:= 15;
            END_IF

		15:
			SC_VstupnyDotlacac.StepName:= '15 - Zasunutie dotlacaca pri poruche';
			SC_VstupnyDotlacac.IdleTime.PT:= T#3s;
			SC_VstupnyDotlacac.AlarmTime.PT:= T#3s;

			Preklapac.OUT.VstupnyDotlacac_VYSUN_YV1:= FALSE;
			Preklapac.OUT.VstupnyDotlacac_ZASUN_YV2:= TRUE;
			Alarmy[5]:= TRUE;
			SC_VstupnyDotlacac.ResetStep:= TRUE;
			SC_VstupnyDotlacac.Step:= 0;

        20:
            SC_VstupnyDotlacac.StepName:= '20 - Zasunutie dotlacaca';
            SC_VstupnyDotlacac.IdleTime.PT:= T#3s;
            SC_VstupnyDotlacac.AlarmTime.PT:= T#3s;

            IF Preklapac.Automat THEN
                SC_VstupnyDotlacac.AlarmTime.IN:= TRUE;
            ELSE
                SC_VstupnyDotlacac.IdleTime.IN:= TRUE;
            END_IF

            IF NOT SC_VstupnyDotlacac.Switch1 THEN
                Preklapac.OUT.VstupnyDotlacac_VYSUN_YV1:= FALSE;
                Preklapac.OUT.VstupnyDotlacac_ZASUN_YV2:= TRUE;
                SC_VstupnyDotlacac.Switch1:= TRUE;
            END_IF

            IF Preklapac.IN.VstupnyDotlacac_ZASUNUTY_MS2 OR SC_VstupnyDotlacac.IdleTime.Q THEN
                SC_VstupnyDotlacac.ResetStep:= TRUE;
                SC_VstupnyDotlacac.Step:= 0;
            ELSIF SC_VstupnyDotlacac.AlarmTime.Q THEN
                Alarmy[6]:= TRUE;
                SC_VstupnyDotlacac.ResetStep:= TRUE;
                SC_VstupnyDotlacac.Step:= 0;
            END_IF

    END_CASE

END_ACTION
```

#### Zdvih.st
```iecst
ACTION Zdvih:

    //Volanie funkcie SequenceControl//
    SequenceControl(SC:= SC_Zdvih);

    CASE SC_Zdvih.Step OF

        0:
            SC_Zdvih.StepName:= '0 - Nulovanie';
            Zdvih_VYSUN:= FALSE;
            Zdvih_ZASUN:= FALSE;
//            Preklapac.OUT.Vytah_ZDVIH_YV5:= FALSE;
//            Preklapac.OUT.Vytah_ZOSTUP_YV6:= FALSE;

            IF SC_Preklapac.Step <> 0 THEN
                SC_Zdvih.ResetStep:= TRUE;
                SC_Zdvih.Step:= 1;
            END_IF

        1:
            SC_Zdvih.StepName:= '1 - Rozhodnutie o cinnosti';
            IF Zdvih_VYSUN THEN
                SC_Zdvih.Step:= 10;
            ELSIF Zdvih_ZASUN THEN
                SC_Zdvih.Step:= 20;
            END_IF

        10:
            SC_Zdvih.StepName:= '10 - Vysunutie zdvihu';
            SC_Zdvih.IdleTime.PT:= T#3s;
            SC_Zdvih.AlarmTime.PT:= T#3s;

            IF Preklapac.Automat THEN
                SC_Zdvih.AlarmTime.IN:= TRUE;
            ELSE
                SC_Zdvih.IdleTime.IN:= TRUE;
            END_IF

            IF NOT SC_Zdvih.Switch1 THEN
                Preklapac.OUT.Vytah_ZOSTUP_YV6:= FALSE;
                Preklapac.OUT.Vytah_ZDVIH_YV5:= TRUE;
                SC_Zdvih.IdleTime.IN:= TRUE;
                SC_Zdvih.Switch1:= TRUE;
            END_IF

            IF Preklapac.IN.Vytah_HornaPoloha_MS5 OR SC_Zdvih.IdleTime.Q THEN
                SC_Zdvih.ResetStep:= TRUE;
                SC_Zdvih.Step:= 0;
            ELSIF SC_Zdvih.AlarmTime.Q THEN
                SC_Zdvih.ResetStep:= TRUE;
                SC_Zdvih.Step:= 15;
            END_IF

		15:
			SC_Zdvih.StepName:= '15 - Zasunutie zdvihu pri poruche';
			SC_Zdvih.IdleTime.PT:= T#3s;
			SC_Zdvih.AlarmTime.PT:= T#3s;

			Preklapac.OUT.Vytah_ZDVIH_YV5:= FALSE;
			Preklapac.OUT.Vytah_ZOSTUP_YV6:= TRUE;
			Alarmy[7]:= TRUE;
			SC_Zdvih.ResetStep:= TRUE;
			SC_Zdvih.Step:= 0;

        20:
            SC_Zdvih.StepName:= '20 - Zasunutie zdvihu';
            SC_Zdvih.IdleTime.PT:= T#3s;
            SC_Zdvih.AlarmTime.PT:= T#3s;

            IF Preklapac.Automat THEN
                SC_Zdvih.AlarmTime.IN:= TRUE;
            ELSE
                SC_Zdvih.IdleTime.IN:= TRUE;
            END_IF

            IF NOT SC_Zdvih.Switch1 THEN
                Preklapac.OUT.Vytah_ZDVIH_YV5:= FALSE;
                Preklapac.OUT.Vytah_ZOSTUP_YV6:= TRUE;
                SC_Zdvih.Switch1:= TRUE;
            END_IF

            IF Preklapac.IN.Vytah_SpodnaPoloha_MS6 OR SC_Zdvih.IdleTime.Q THEN
                SC_Zdvih.ResetStep:= TRUE;
                SC_Zdvih.Step:= 0;
            ELSIF SC_Zdvih.AlarmTime.Q THEN
                Alarmy[8]:= TRUE;
                SC_Zdvih.ResetStep:= TRUE;
                SC_Zdvih.Step:= 0;
            END_IF

    END_CASE

END_ACTION
```

#### VystupnyDotlacac.st
```iecst
ACTION VystupnyDotlacac:

    //Volanie funkcie SequenceControl//
    SequenceControl(SC:= SC_VystupnyDotlacac);

    CASE SC_VystupnyDotlacac.Step OF

        0:
            SC_VystupnyDotlacac.StepName:= '0 - Nulovanie';
            VystupnyDotlacac_VYSUN:= FALSE;
            VystupnyDotlacac_ZASUN:= FALSE;
            (*Preklapac.OUT.VystupnyDotlacac_VYSUN_YV3:= FALSE;*)

            IF SC_Preklapac.Step <> 0 THEN
                SC_VystupnyDotlacac.ResetStep:= TRUE;
                SC_VystupnyDotlacac.Step:= 1;
            END_IF

        1:
            SC_VystupnyDotlacac.StepName:= '1 - Rozhodnutie o cinnosti';
            IF VystupnyDotlacac_VYSUN THEN
                SC_VystupnyDotlacac.Step:= 10;
            ELSIF VystupnyDotlacac_ZASUN THEN
                SC_VystupnyDotlacac.Step:= 20;
            END_IF

        10:
            SC_VystupnyDotlacac.StepName:= '10 - Vysunutie dotlacaca';
            SC_VystupnyDotlacac.IdleTime.PT:= T#3s;
            SC_VystupnyDotlacac.AlarmTime.PT:= T#3s;

            IF Preklapac.Automat THEN
                SC_VystupnyDotlacac.AlarmTime.IN:= TRUE;
            ELSE
                SC_VystupnyDotlacac.IdleTime.IN:= TRUE;
            END_IF

            IF NOT SC_VystupnyDotlacac.Switch1 THEN
                Preklapac.OUT.VystupnyDotlacac_VYSUN_YV3:= TRUE;
                SC_VystupnyDotlacac.IdleTime.IN:= TRUE;
                SC_VystupnyDotlacac.Switch1:= TRUE;
            END_IF

            IF Preklapac.IN.VystupnyDotlacac_VYSUNUTY_MS3 OR SC_VystupnyDotlacac.IdleTime.Q THEN
                SC_VystupnyDotlacac.ResetStep:= TRUE;
                SC_VystupnyDotlacac.Step:= 0;
            ELSIF SC_VystupnyDotlacac.AlarmTime.Q THEN
                SC_VystupnyDotlacac.ResetStep:= TRUE;
                SC_VystupnyDotlacac.Step:= 15;
            END_IF

		15:
			SC_VystupnyDotlacac.StepName:= '15 - Zasunutie dotlacaca pri poruche';
			SC_VystupnyDotlacac.IdleTime.PT:= T#3s;
			SC_VystupnyDotlacac.AlarmTime.PT:= T#3s;

			Preklapac.OUT.VystupnyDotlacac_VYSUN_YV3:= FALSE;
			Alarmy[9]:= TRUE;
			SC_VystupnyDotlacac.ResetStep:= TRUE;
			SC_VystupnyDotlacac.Step:= 0;

        20:
            SC_VystupnyDotlacac.StepName:= '20 - Zasunutie dotlacaca';
            SC_VystupnyDotlacac.IdleTime.PT:= T#3s;
            SC_VystupnyDotlacac.AlarmTime.PT:= T#3s;

            IF Preklapac.Automat THEN
                SC_VystupnyDotlacac.AlarmTime.IN:= TRUE;
            ELSE
                SC_VystupnyDotlacac.IdleTime.IN:= TRUE;
            END_IF

            IF NOT SC_VystupnyDotlacac.Switch1 THEN
                Preklapac.OUT.VystupnyDotlacac_VYSUN_YV3:= FALSE;
                SC_VystupnyDotlacac.Switch1:= TRUE;
            END_IF

            IF Preklapac.IN.VystupnyDotlacac_ZASUNUTY_MS4 OR SC_VystupnyDotlacac.IdleTime.Q THEN
                SC_VystupnyDotlacac.ResetStep:= TRUE;
                SC_VystupnyDotlacac.Step:= 0;
            ELSIF SC_VystupnyDotlacac.AlarmTime.Q THEN
                Alarmy[10]:= TRUE;
                SC_VystupnyDotlacac.ResetStep:= TRUE;
                SC_VystupnyDotlacac.Step:= 0;
            END_IF

    END_CASE

END_ACTION
```

### Program Logical/Program/Alarmy (IEC)

#### Main.st - Init, cyclic, exit code
```iecst
PROGRAM _INIT
	(* Insert code here *)

END_PROGRAM

PROGRAM _CYCLIC

    //Alarmy pracoviska//
    //A0 - Porucha tlaku vzduchu !!!
    //A1 - Porucha PLC karty AB2 - CAN Slave !!!
    //A2 - Porucha PLC karty AB3 - Digitálne Vstupy !!!
    //A3 - Porucha PLC karty AB4 - Digitálne Vystupy !!!
    //A4 - Porucha bezpecnostného okruhu !!!
    //A5 - Porucha vysunutia vstupného dotlácaca !!!
    //A6 - Porucha zasunutia vstupného dotlácaca !!!
    //A7 - Porucha zdvihu vytahu !!!
    //A8 - Porucha zostupu vytahu !!!
    //A9 - Porucha vysunutia vystupneho dotlacaca !!!
    //A10 - Porucha zasunutia vystupneho dotlacaca !!!

    //***********************************Hladanie poruchy*****************************************//

    FOR a:=0 TO 100 BY 1 DO
        Alarmy[a];
        IF Alarmy[a] = TRUE THEN
            NastalaPorucha:= TRUE;
        END_IF
    END_FOR

    //********************************Zobrazenie symbolu alarmu*****************************************************//

    IF NastalaPorucha THEN
        Vizu.ZobrazSymbolAlarmu:= Blikac500ms;
    ELSE
        Vizu.ZobrazSymbolAlarmu:= FALSE;
    END_IF

    //*************************************Potvrdenie alarmov*********************************************************//
    IF PotvrdenieAlarmov THEN
        brsmemset(ADR(Alarmy),0,SIZEOF(Alarmy));
        NastalaPorucha:= FALSE;
        Zariadenie.Majak_HukackaON:= FALSE;
        PotvrdenieAlarmov:= FALSE;
    END_IF

    //**************************************Porucha tlaku vzduchu*********************************************************//
    CasKontroly_TlakuVzduchu.IN:= Zariadenie.IN.Safety_Aktivne AND NOT Zariadenie.IN.TlakVzduchu_OK_S1;

    IF CasKontroly_TlakuVzduchu.Q THEN
        Alarmy[0]:= TRUE;
    END_IF

    CasKontroly_TlakuVzduchu.PT:= T#2s;
    CasKontroly_TlakuVzduchu();

    //**********************************Porucha - karty PLC niesu online**************************************************//
    CasKontroly_KarietPLC.IN:= Zariadenie.IN.Safety_Aktivne AND NOT Zariadenie.STAV.Hardware_OK;

    IF CasKontroly_KarietPLC.Q THEN
        IF NOT Hardware.KartaAB2_CANSlave_OK THEN
            Alarmy[1]:= TRUE;
        END_IF
        IF NOT Hardware.KartaAB3_16DI_OK THEN
            Alarmy[2]:= TRUE;
        END_IF
        IF NOT Hardware.KartaAB4_16DO_OK THEN
            Alarmy[3]:= TRUE;
        END_IF
    END_IF

    CasKontroly_KarietPLC.PT:= T#2s;
    CasKontroly_KarietPLC();

    //*********************************Porucha - bezpečnostného okruhu*******************************************************//
//    IF EDGENEG(Zariadenie.IN.Safety_Aktivne) THEN
//        Alarmy[4]:= TRUE;
//    END_IF

END_PROGRAM

PROGRAM _EXIT
	(* Insert code here *)

END_PROGRAM
```

#### Variables.var - Local variables
```iecst
VAR
	a : USINT := 0;
	CasKontroly_KarietPLC : TON;
	CasKontroly_TlakuVzduchu : TON;
END_VAR
```

### Program Logical/HMI/OvladanieVizu (IEC)

#### Main.st - Init, cyclic, exit code
```iecst
PROGRAM _INIT
	CasZobrazeniaUvodnejObrazovky.IN:= TRUE;

END_PROGRAM

PROGRAM _CYCLIC

    //*********************************************Zobrazenie úvodnej obrazovky**********************************************//
    IF NOT CasZobrazeniaUvodnejObrazovky.Q THEN
        Vizu.CisloZadanejObrazovky:= 0;
        IF EDGEPOS (Blikac500ms = TRUE) THEN
            IF Vizu.Slider < 30 THEN
                Vizu.Slider:= Vizu.Slider+1;
            ELSE
                Vizu.Slider:= 0;
            END_IF
        END_IF
    END_IF

    CasZobrazeniaUvodnejObrazovky.PT:= T#20s;
    CasZobrazeniaUvodnejObrazovky();

    //******************************************************Podsvietenie tlačítok**********************************************************//
    //Tlačítko Reset CS//
    IF Zariadenie.IN.Safety_SpatnaVazba_KF1 AND NOT Zariadenie.IN.Safety_Aktivne THEN
        Vizu.PodsvietenieTlacitka_ResetCS:= Blikac500ms;
    ELSIF Zariadenie.IN.Safety_Aktivne THEN
        Vizu.PodsvietenieTlacitka_ResetCS:= 2;
    ELSE
        Vizu.PodsvietenieTlacitka_ResetCS:= 3;
    END_IF

    //Tlačítko alarmy//
    IF NastalaPorucha THEN
        Vizu.FarbaTlacitkaAlarm_Index:= Blikac500ms;
    ELSE
        Vizu.FarbaTlacitkaAlarm_Index:= FALSE;
    END_IF

    //************************************Prepnutie na obrazovku Automatického režimu******************************************//
    IF EDGEPOS (CasZobrazeniaUvodnejObrazovky.Q = TRUE) THEN
        Vizu.CisloZadanejObrazovky:= 2;
    END_IF

    //*************************************************Zamknutie tlačítok*******************************************************//
    //Tlačítko režim manual//
    IF Zariadenie.STAV.Automat THEN
		Vizu.TL_RezimManual_DISABLE:= TRUE;
	ELSIF NOT Zariadenie.IN.Safety_Aktivne THEN
		Vizu.TL_RezimManual_DISABLE:= TRUE;
    ELSE
        Vizu.TL_RezimManual_DISABLE:= FALSE;
    END_IF

    //Tlačítko Štart Automat//
    IF NOT Zariadenie.IN.Safety_Aktivne THEN
        Vizu.TL_StartAutomat_DISABLE:= TRUE;
    ELSIF NastalaPorucha THEN
        Vizu.TL_StartAutomat_DISABLE:= TRUE;
    ELSIF NOT Zariadenie.STAV.READY_TO_START THEN
        Vizu.TL_StartAutomat_DISABLE:= TRUE;
    ELSIF Zariadenie.STAV.Automat THEN
		Vizu.TL_StartAutomat_DISABLE:= TRUE;
	ELSIF NOT Preklapac.IN.VystupnyDopravnik_StavOK THEN
		Vizu.TL_StartAutomat_DISABLE:= TRUE;
    ELSE
        Vizu.TL_StartAutomat_DISABLE:= FALSE;
    END_IF

    //Tlačítko Ukončenie cyklu//
    IF Zariadenie.STAV.PoINIT THEN
        Vizu.TL_UkoncenieCyklu_DISABLE:= FALSE;
    ELSE
        Vizu.TL_UkoncenieCyklu_DISABLE:= TRUE;
    END_IF

    //Tlačítko Reset//
    IF Zariadenie.STAV.PoINIT AND NOT Zariadenie.STAV.UkoncenieCyklu_BUSY THEN
        Vizu.TL_Reset_DISABLE:= TRUE;
    ELSE
        Vizu.TL_Reset_DISABLE:= FALSE;
    END_IF

    //Tlačítka ovládania preklápača v ručnom režime//
    //Dotláčače//
    IF NOT Zariadenie.IN.Safety_Aktivne THEN
        Vizu.TL_RR_PreklapacDotlacace_DISABLE:= TRUE;
    ELSIF NastalaPorucha THEN
        Vizu.TL_RR_PreklapacDotlacace_DISABLE:= TRUE;
    ELSE
        Vizu.TL_RR_PreklapacDotlacace_DISABLE:= FALSE;
    END_IF

    //Zdvih//
    IF NOT Zariadenie.IN.Safety_Aktivne THEN
        Vizu.TL_RR_PreklapacZdvih_DISABLE:= TRUE;
    ELSIF NastalaPorucha THEN
        Vizu.TL_RR_PreklapacZdvih_DISABLE:= TRUE;
    ELSIF NOT Preklapac.IN.VystupnyDotlacac_ZASUNUTY_MS4 THEN
        Vizu.TL_RR_PreklapacZdvih_DISABLE:= TRUE;
    ELSE
        Vizu.TL_RR_PreklapacZdvih_DISABLE:= FALSE;
    END_IF

	//***************************************************Zobrazenie Pop Up********************************************************//
	IF NOT Preklapac.IN.VystupnyDopravnik_StavOK THEN
		Vizu.TP_PopUp_VystupDopRozpojeny:= 0;
	ELSE
		Vizu.TP_PopUp_VystupDopRozpojeny:= 1;
	END_IF

END_PROGRAM

PROGRAM _EXIT
	(* Insert code here *)

END_PROGRAM
```

#### Variables.var - Local variables
```iecst
VAR
	CasZobrazeniaUvodnejObrazovky : TON := (0);
END_VAR
```

- Visualisation Logical/HMI/Visu (not shown)

### Program Logical/Blikace/Blikanie100ms (IEC)

#### Blikanie100ms.st - Init, cyclic, exit code
```iecst
PROGRAM _INIT
	(* Insert code here *)

END_PROGRAM

PROGRAM _CYCLIC

	IF NOT Blikac100ms THEN
		Blikac100ms:= TRUE;
	ELSE
		Blikac100ms:= FALSE;
	END_IF

END_PROGRAM

PROGRAM _EXIT
	(* Insert code here *)

END_PROGRAM
```

### Program Logical/Blikace/Blikanie200ms (IEC)

#### Blikanie200ms.st - Init, cyclic, exit code
```iecst
PROGRAM _INIT
	(* Insert code here *)

END_PROGRAM

PROGRAM _CYCLIC

	IF NOT Blikac200ms THEN
		Blikac200ms:= TRUE;
	ELSE
		Blikac200ms:= FALSE;
	END_IF

END_PROGRAM

PROGRAM _EXIT
	(* Insert code here *)

END_PROGRAM
```

### Program Logical/Blikace/Blikanie500ms (IEC)

#### Blikanie500ms.st - Init, cyclic, exit code
```iecst
PROGRAM _INIT
	(* Insert code here *)

END_PROGRAM

PROGRAM _CYCLIC
	IF NOT Blikac500ms THEN
		Blikac500ms:= TRUE;
	ELSE
		Blikac500ms:= FALSE;
	END_IF

END_PROGRAM

PROGRAM _EXIT
	(* Insert code here *)

END_PROGRAM
```

### Program Logical/Blikace/Blikanie1s (IEC)

#### Blikanie1s.st - Init, cyclic, exit code
```iecst
PROGRAM _INIT
	(* Insert code here *)

END_PROGRAM

PROGRAM _CYCLIC
	IF NOT Blikac1s THEN
		Blikac1s:= TRUE;
	ELSE
		Blikac1s:= FALSE;
	END_IF

END_PROGRAM

PROGRAM _EXIT
	(* Insert code here *)

END_PROGRAM
```

### DatumCasGlobal.var
```iecst
VAR
	PLC_Cas : PLC_Cas_typ;
	PLC_Datum : PLC_Datum_typ;
	Sekunda_STR : STRING[2];
	Minuta_STR : STRING[2];
	Hodina_STR : STRING[2];
	Den_STR : STRING[2];
	Mesiac_STR : STRING[2];
	Rok_STR_4_Znaky : STRING[4];
	Rok_STR_2_Znaky : STRING[2];
END_VAR
```

### DatumCasGlobal.typ
```iecst
TYPE
	PLC_Cas_typ : 	STRUCT
		Sekundy : USINT;
		Minuty : USINT;
		Hodiny : USINT;
	END_STRUCT;
	PLC_Datum_typ : 	STRUCT
		Den : USINT;
		Mesiac : USINT;
		Rok : UINT;
	END_STRUCT;
END_TYPE
```

### Program Logical/DatumCasPLC/DatumCasPLC (IEC)

#### Main.st - Init, cyclic, exit code
```iecst
PROGRAM _INIT
	(* Insert code here *)

END_PROGRAM

PROGRAM _CYCLIC

	//Vyčítavanie systémového času//
	DTGetTime_1.enable:= TRUE;
	DTGetTime_1();
	DT_TO_DTStructure(DTGetTime_1.DT1,ADR(PLC_DatumCas));

	PLC_Cas.Sekundy:= PLC_DatumCas.second;
	PLC_Cas.Minuty:= PLC_DatumCas.minute;
	PLC_Cas.Hodiny:= PLC_DatumCas.hour;

	PLC_Datum.Den:= PLC_DatumCas.day;
	PLC_Datum.Mesiac:= PLC_DatumCas.month;
	PLC_Datum.Rok:= PLC_DatumCas.year;

	//Prevod času na String//
	//Sekundy//
	IF PLC_Cas.Sekundy < 10 THEN
		Sekundy_String:= USINT_TO_STRING(PLC_Cas.Sekundy);
		Sekunda_STR:= '0';
		brsstrcat(ADR(Sekunda_STR),ADR(Sekundy_String));
	ELSE
		Sekunda_STR:= USINT_TO_STRING(PLC_Cas.Sekundy);
	END_IF

	//Minuty//
	IF PLC_Cas.Minuty < 10 THEN
		Minuty_String:= USINT_TO_STRING(PLC_Cas.Minuty);
		Minuta_STR:= '0';
		brsstrcat(ADR(Minuta_STR),ADR(Minuty_String));
	ELSE
		Minuta_STR:= USINT_TO_STRING(PLC_Cas.Minuty);
	END_IF

	//Hodiny//
	IF PLC_Cas.Hodiny < 10 THEN
		Hodiny_String:= USINT_TO_STRING(PLC_Cas.Hodiny);
		Hodina_STR:= '0';
		brsstrcat(ADR(Hodina_STR),ADR(Hodiny_String));
	ELSE
		Hodina_STR:= USINT_TO_STRING(PLC_Cas.Hodiny);
	END_IF

	//Prevod dátumu na String//
	//Deň//
	IF PLC_Datum.Den < 10 THEN
		Den_String:= USINT_TO_STRING(PLC_Datum.Den);
		Den_STR:= '0';
		brsstrcat(ADR(Den_STR),ADR(Den_String));
	ELSE
		Den_STR:= USINT_TO_STRING(PLC_Datum.Den);
	END_IF

	//Masiac//
	IF PLC_Datum.Mesiac < 10 THEN
		Mesiac_String:= USINT_TO_STRING(PLC_Datum.Mesiac);
		Mesiac_STR:= '0';
		brsstrcat(ADR(Mesiac_STR),ADR(Mesiac_String));
	ELSE
		Mesiac_STR:= USINT_TO_STRING(PLC_Datum.Mesiac);
	END_IF

	//Rok - 4 znaky//
	Rok_STR_4_Znaky:= UINT_TO_STRING(PLC_Datum.Rok);

	//Rok - posledné 2 znaky//
	length := brsstrlen(ADR(Rok_STR_4_Znaky)); //Zistí počet znakov//

	IF length >= 4 THEN
		brsmemcpy(ADR(PoleUSINT),ADR(Rok_STR_4_Znaky),SIZEOF(Rok_STR_4_Znaky));
		i := PoleUSINT[length-2]; //Vyčítanie predposledného znaku//
		brsstrcpy(ADR(DvaZnaky),ADR(i));
		i := PoleUSINT[length-1]; //Vyčítanie posledneho znaku//
		brsstrcat(ADR(DvaZnaky),ADR(i));
	END_IF

	Rok_STR_2_Znaky:= DvaZnaky;

END_PROGRAM

PROGRAM _EXIT
	(* Insert code here *)

END_PROGRAM
```

#### Variables.var - Local variables
```iecst
VAR
	PLC_DatumCas : DTStructure;
	DTGetTime_1 : DTGetTime;
	Sekundy_String : STRING[2];
	Minuty_String : STRING[2];
	Hodiny_String : STRING[2];
	Den_String : STRING[2];
	Mesiac_String : STRING[2];
	length : UDINT;
	PoleUSINT : ARRAY[0..3] OF USINT;
	i : USINT;
	DvaZnaky : STRING[2];
END_VAR
```
